PROGRAM Constants
VAR
	
	bInit:BOOL:=TRUE;

END_VAR

IF bInit THEN
	bInit:=FALSE;
	//Lighting Init
	Topic.stBuilding.stFloorOne.stLights.stLighting.aModes[0]:='Automatic';
	Topic.stBuilding.stFloorOne.stLights.stLighting.aModes[1]:='Manual';
	Topic.stBuilding.stFloorOne.stLights.stLighting.sMode:='Init';
END_IF

END_PROGRAM

(* stored: Version 1.1.0.1, ProductVersion 3.1.4024.12
   POU Constants: Id {3cd51791-fad7-404a-90f7-f0bee9d96ece}, SpecialFunc None *)
